// SIMATIC STEP 7 (V5.x) project PROBLEM 6
// CPU: CPU 314C-2 DP
// station: Hardware
// station: SIMATIC 300(1)
// station: P_ADR_BUS
// program: S7 Program(1)

SYMBOL_TABLE
"3S PASSED"	M 1.1	BOOL
"6S PASSED"	M 1.2	BOOL
"STATE 1"	M 3.1	BOOL
"STATE 2"	M 3.2	BOOL
END_SYMBOL_TABLE

ORGANIZATION_BLOCK OB 1
TITLE = "Main Program Sweep (Cycle)"
//PROBLEM 6
VERSION : 0.1
VAR_TEMP
  OB1_EV_CLASS : BYTE ;	//Bits 0-3 = 1 (Coming event), Bits 4-7 = 1 (Event class 1)
  OB1_SCAN_1 : BYTE ;	//1 (Cold restart scan 1 of OB 1), 3 (Scan 2-n of OB 1)
  OB1_PRIORITY : BYTE ;	//Priority of OB Execution
  OB1_OB_NUMBR : BYTE ;	//1 (Organization block 1, OB1)
  OB1_RESERVED_1 : BYTE ;	//Reserved for system
  OB1_RESERVED_2 : BYTE ;	//Reserved for system
  OB1_PREV_CYCLE : INT ;	//Cycle time of previous OB1 scan (milliseconds)
  OB1_MIN_CYCLE : INT ;	//Minimum cycle time of OB1 (milliseconds)
  OB1_MAX_CYCLE : INT ;	//Maximum cycle time of OB1 (milliseconds)
  OB1_DATE_TIME : DATE_AND_TIME ;	//Date and time OB1 started
END_VAR
BEGIN
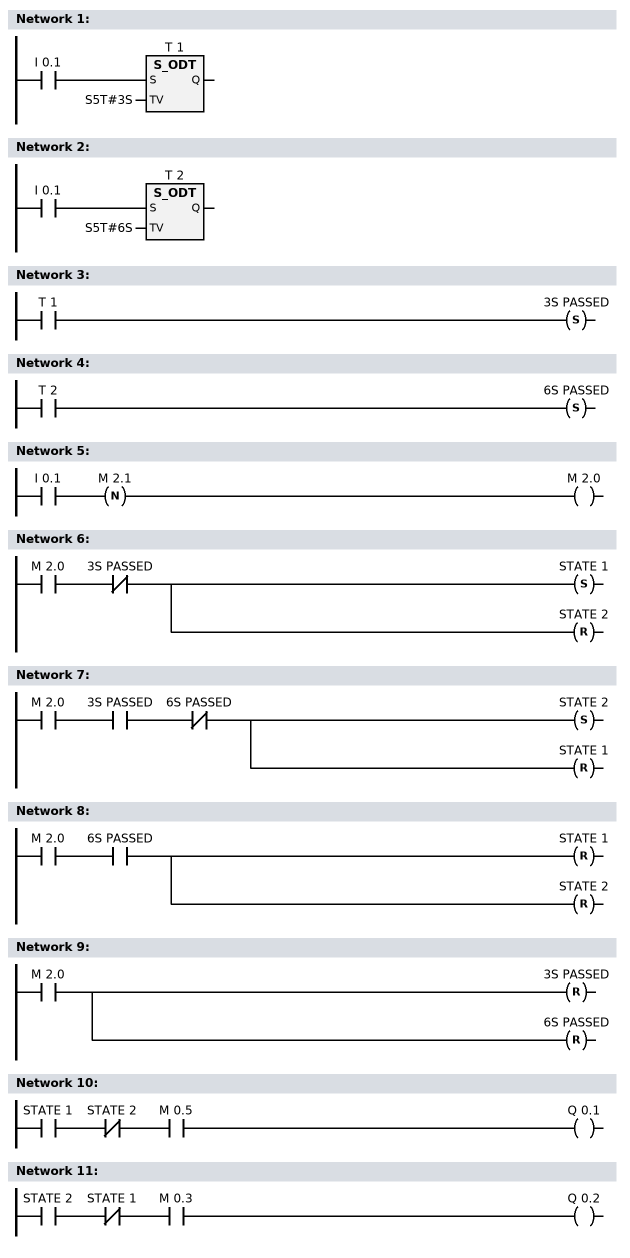
NETWORK
TITLE =
      A     I 0.1;
      L     S5T#3S;
      SD    T 1;
      NOP   0;
      NOP   0;
      NOP   0;
      NOP   0;
NETWORK
TITLE =
      A     I 0.1;
      L     S5T#6S;
      SD    T 2;
      NOP   0;
      NOP   0;
      NOP   0;
      NOP   0;
NETWORK
TITLE =
      A     T 1;
      S     "3S PASSED";
NETWORK
TITLE =
      A     T 2;
      S     "6S PASSED";
NETWORK
TITLE =
      A     I 0.1;
      FN    M 2.1;
      =     M 2.0;
NETWORK
TITLE =
      A     M 2.0;
      AN    "3S PASSED";
      S     "STATE 1";
      R     "STATE 2";
NETWORK
TITLE =
      A     M 2.0;
      A     "3S PASSED";
      AN    "6S PASSED";
      S     "STATE 2";
      R     "STATE 1";
NETWORK
TITLE =
      A     M 2.0;
      A     "6S PASSED";
      R     "STATE 1";
      R     "STATE 2";
NETWORK
TITLE =
      A     M 2.0;
      R     "3S PASSED";
      R     "6S PASSED";
NETWORK
TITLE =
      A     "STATE 1";
      AN    "STATE 2";
      A     M 0.5;
      =     Q 0.1;
NETWORK
TITLE =
      A     "STATE 2";
      AN    "STATE 1";
      A     M 0.3;
      =     Q 0.2;
END_ORGANIZATION_BLOCK
